// TIA Portal V16 export
// export: Created 2021-09-01T08:19:44.7263229Z, ExportSetting WithDefaults, DisplayName Totally Integrated Automation Portal, DisplayVersion V16 Update 3, DisplayName TIA Portal Version Control Interface, DisplayVersion V16 Update 2, DisplayName TIA Portal Openness, DisplayVersion V16 Update 3, DisplayName TIA Portal Teamcenter Gateway, DisplayVersion V16, DisplayName STEP 7 Professional, DisplayVersion V16 Update 3, DisplayName STEP 7 Safety, DisplayVersion V16, DisplayName WinCC Advanced, DisplayVersion V16 Update 3
FUNCTION_BLOCK "AllPump"   // FB2, FBD
{ S7_Optimized_Access := 'TRUE' }
VERSION : 0.1
// stored: AutoNumber true, IsIECCheckEnabled false, IsRetainMemResEnabled false, MemoryReserve 100, SetENOAutomatically false, UDAEnableTagReadback false
   VAR
      PU30x { S7_SetPoint := 'True'} : "PumpCntrl2Pu1Fc";
      cmUZ1 { S7_SetPoint := 'True'} : Bool;
      tmrLowPresP30x { S7_SetPoint := 'True'} : TON_TIME;
      tmrLowFreqP30x { S7_SetPoint := 'True'} : TON_TIME;
      tLowPresP30x { S7_SetPoint := 'True'} : Time;
      tLowFreqP30x : Time;
   END_VAR
BEGIN

REGION Network 1: P30x - выбор рабочего
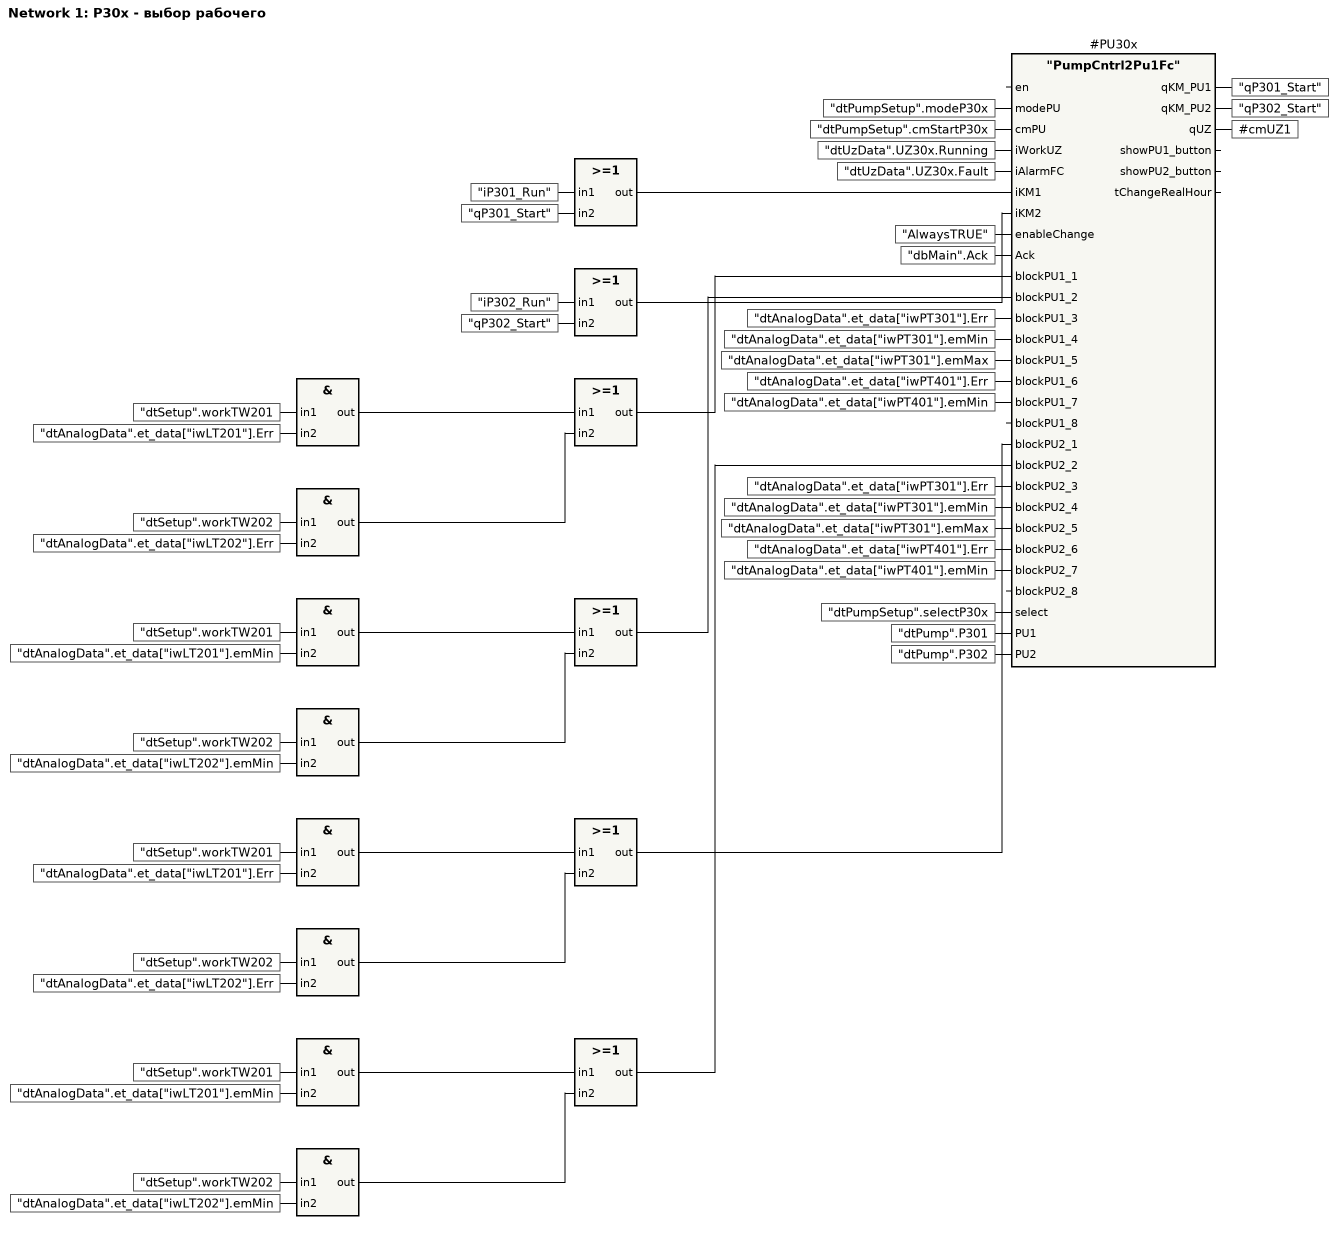
   #PU30x(modePU := "dtPumpSetup".modeP30x,   // "PumpCntrl2Pu1Fc"
          cmPU := "dtPumpSetup".cmStartP30x,
          iWorkUZ := "dtUzData".UZ30x.Running,
          iAlarmFC := "dtUzData".UZ30x.Fault,
          iKM1 := "iP301_Run" OR "qP301_Start",
          iKM2 := "iP302_Run" OR "qP302_Start",
          enableChange := "AlwaysTRUE",
          Ack := "dbMain".Ack,
          blockPU1_1 := ("dtSetup".workTW201 AND "dtAnalogData".et_data["iwLT201"].Err) OR ("dtSetup".workTW202 AND "dtAnalogData".et_data["iwLT202"].Err),
          blockPU1_2 := ("dtSetup".workTW201 AND "dtAnalogData".et_data["iwLT201"].emMin) OR ("dtSetup".workTW202 AND "dtAnalogData".et_data["iwLT202"].emMin),
          blockPU1_3 := "dtAnalogData".et_data["iwPT301"].Err,
          blockPU1_4 := "dtAnalogData".et_data["iwPT301"].emMin,
          blockPU1_5 := "dtAnalogData".et_data["iwPT301"].emMax,
          blockPU1_6 := "dtAnalogData".et_data["iwPT401"].Err,
          blockPU1_7 := "dtAnalogData".et_data["iwPT401"].emMin,
          blockPU2_1 := ("dtSetup".workTW201 AND "dtAnalogData".et_data["iwLT201"].Err) OR ("dtSetup".workTW202 AND "dtAnalogData".et_data["iwLT202"].Err),
          blockPU2_2 := ("dtSetup".workTW201 AND "dtAnalogData".et_data["iwLT201"].emMin) OR ("dtSetup".workTW202 AND "dtAnalogData".et_data["iwLT202"].emMin),
          blockPU2_3 := "dtAnalogData".et_data["iwPT301"].Err,
          blockPU2_4 := "dtAnalogData".et_data["iwPT301"].emMin,
          blockPU2_5 := "dtAnalogData".et_data["iwPT301"].emMax,
          blockPU2_6 := "dtAnalogData".et_data["iwPT401"].Err,
          blockPU2_7 := "dtAnalogData".et_data["iwPT401"].emMin,
          select := "dtPumpSetup".selectP30x,
          PU1 := "dtPump".P301,
          PU2 := "dtPump".P302,
          qKM_PU1 => "qP301_Start",
          qKM_PU2 => "qP302_Start",
          qUZ => #cmUZ1);
END_REGION

REGION Network 2: P30x - частотник
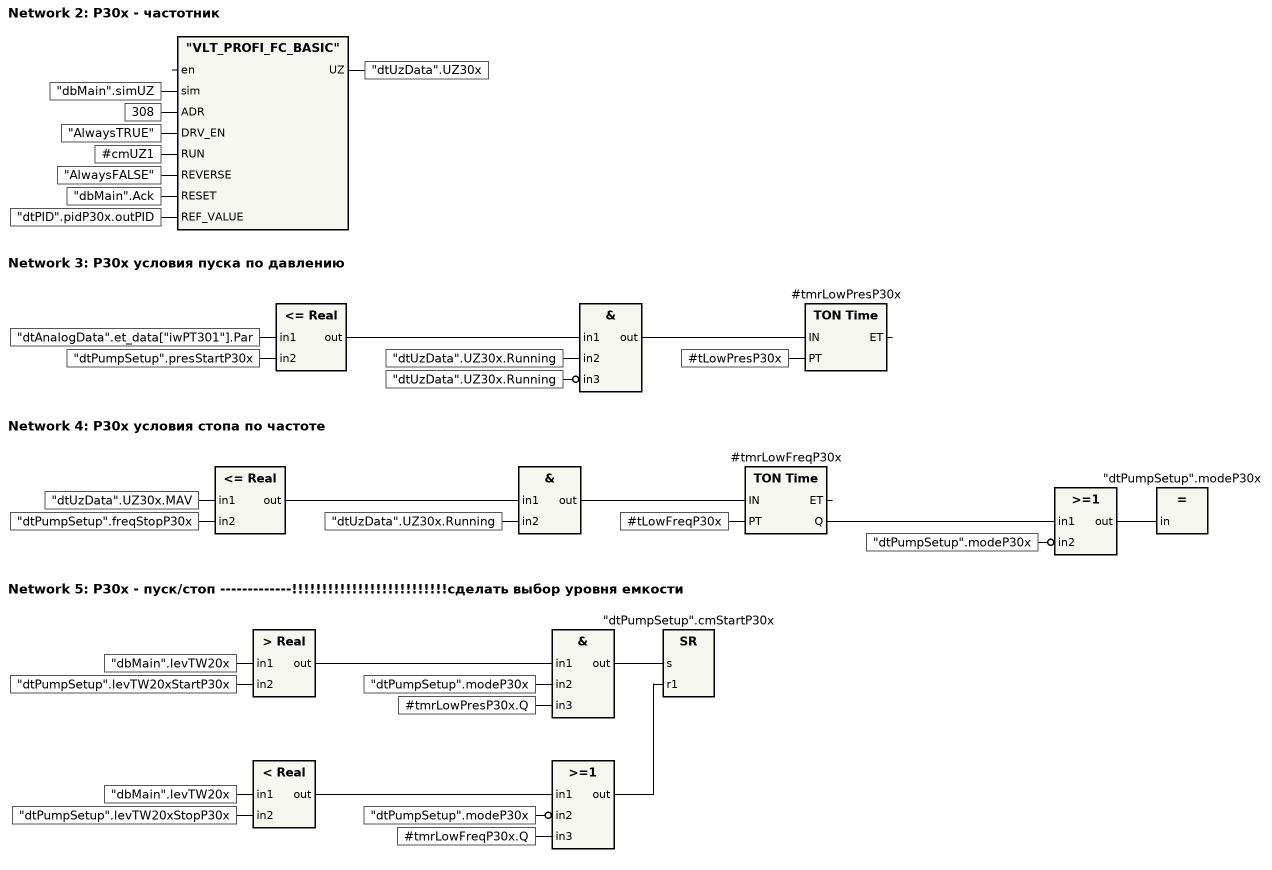
   "VLT_PROFI_FC_BASIC"(sim := "dbMain".simUZ,
                        ADR := 308,
                        DRV_EN := "AlwaysTRUE",
                        RUN := #cmUZ1,
                        REVERSE := "AlwaysFALSE",
                        RESET := "dbMain".Ack,
                        REF_VALUE := "dtPID".pidP30x.outPID,
                        UZ => "dtUzData".UZ30x);
END_REGION

REGION Network 3: P30x условия пуска по давлению
   #tmrLowPresP30x(IN := ("dtAnalogData".et_data["iwPT301"].Par <= "dtPumpSetup".presStartP30x) AND "dtUzData".UZ30x.Running AND NOT "dtUzData".UZ30x.Running,   // TON
                   PT := #tLowPresP30x);
END_REGION

REGION Network 4: P30x условия стопа по частоте
   #tmrLowFreqP30x(IN := ("dtUzData".UZ30x.MAV <= "dtPumpSetup".freqStopP30x) AND "dtUzData".UZ30x.Running,   // TON
                   PT := #tLowFreqP30x);
   "dtPumpSetup".modeP30x := #tmrLowFreqP30x.Q OR NOT "dtPumpSetup".modeP30x;
END_REGION

REGION Network 5: P30x - пуск/стоп -------------!!!!!!!!!!!!!!!!!!!!!!!!!!сделать выбор уровня емкости
   IF ("dbMain".levTW20x > "dtPumpSetup".levTW20xStartP30x) AND "dtPumpSetup".modeP30x AND #tmrLowPresP30x.Q THEN
       "dtPumpSetup".cmStartP30x := TRUE;   // SR flip-flop
   END_IF;
   IF ("dbMain".levTW20x < "dtPumpSetup".levTW20xStopP30x) OR NOT "dtPumpSetup".modeP30x OR #tmrLowFreqP30x.Q THEN
       "dtPumpSetup".cmStartP30x := FALSE;
   END_IF;
END_REGION
END_FUNCTION_BLOCK
